FUNCTION F_Get_Seq_Status : BOOL
VAR_INPUT
	i_seq_sts : BYTE;
END_VAR
VAR_OUTPUT
	o_seq_sts : ST_Sequence_Sts;
END_VAR

o_seq_sts.not_started 		:= i_seq_sts = 0;
o_seq_sts.started 			:= i_seq_sts = 1;
o_seq_sts.completed 		:= i_seq_sts = 2;
o_seq_sts.error 			:= i_seq_sts = 9;

END_FUNCTION

(* stored: Version 1.1.0.1, ProductVersion 3.1.4024.12
   POU F_Get_Seq_Status: Id {a796d6b9-2886-4e9f-95be-12f80c6ae7f8}, SpecialFunc None *)
